// Mitsubishi GX Works2 project: blood pressure test   PLC: FX3G

// global labels: Global1
VAR_GLOBAL
  start_machine AT X007 : BOOL;
  take_test AT X000 : BOOL;
  took_pill AT X001 : BOOL;
  timer_for_gap AT TS1 : BOOL;
  first_test AT D8280 : INT;
  second_test AT D8281 : INT;
  machine_on AT Y007 : BOOL;
  high_blood_pressure AT Y002 : BOOL;
  time_for_next_test AT Y004 : BOOL;
END_VAR
VAR_GLOBAL CONSTANT
  time_to_wait : INT := 50;
END_VAR
VAR_GLOBAL
  took_first_test AT M0 : BOOL;
  test_finish AT M1 : BOOL;
  end_plan AT X006 : BOOL;
  timer AT TC1 : BOOL;
END_VAR
VAR_GLOBAL CONSTANT
  high : INT := 3200;  (* ד *)
END_VAR
VAR_GLOBAL
  hold_light AT M2 : BOOL;
END_VAR

// task Task_01 (event TRUE, interval 0, priority 31): POU_01

PROGRAM POU_01
(* structured ladder/FBD written out as ST: instructions are called as NAME(EN, inputs, outputs); _pN, _eN, _tN stand for wires *)
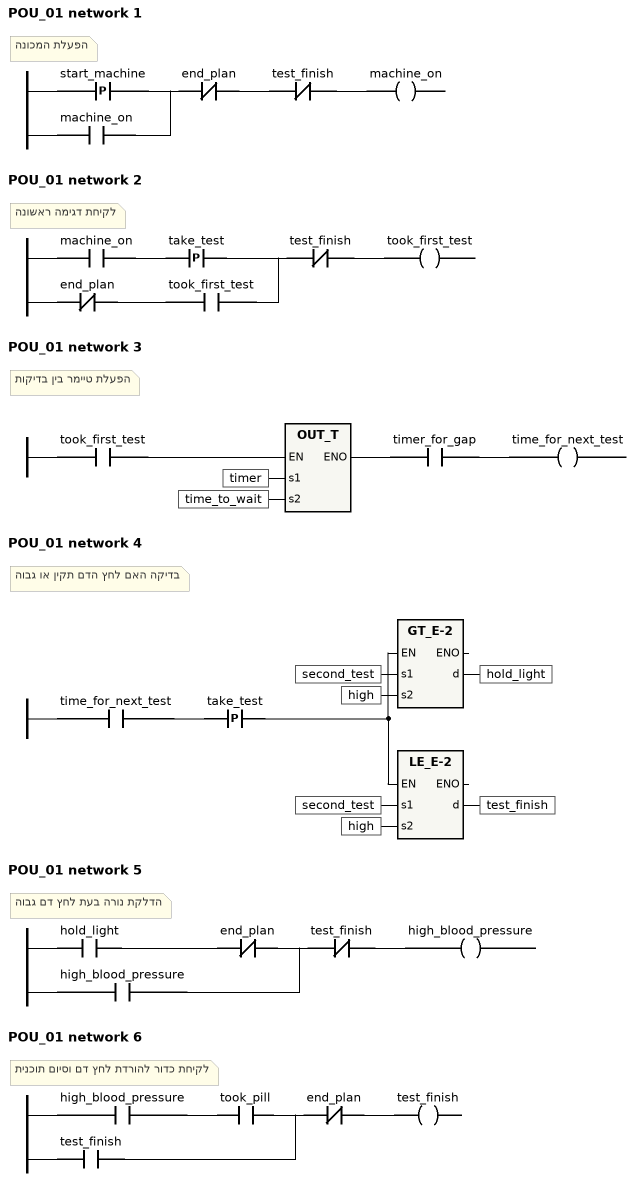
(* network 1 *)
(* הפעלת המכונה *)
machine_on := ((LDP(TRUE, start_machine) OR machine_on) AND NOT end_plan) AND NOT test_finish;
(* network 2 *)
(* לקיחת דגימה ראשונה *)
took_first_test := ((machine_on AND LDP(TRUE, take_test)) OR (NOT end_plan AND took_first_test)) AND NOT test_finish;
(* network 3 *)
(* הפעלת טיימר בין בדיקות *)
_e1 := OUT_T(took_first_test, timer, time_to_wait);
time_for_next_test := _e1 AND timer_for_gap;
(* network 4 *)
(* בדיקה האם לחץ הדם תקין או גבוה *)
_p1 := time_for_next_test AND LDP(TRUE, take_test);
GT_E(_p1, second_test, high, hold_light);
LE_E(_p1, second_test, high, test_finish);
(* network 5 *)
(* הדלקת נורה בעת לחץ דם גבוה *)
high_blood_pressure := ((hold_light AND NOT end_plan) OR high_blood_pressure) AND NOT test_finish;
(* network 6 *)
(* לקיחת כדור להורדת לחץ דם וסיום תוכנית *)
test_finish := ((high_blood_pressure AND took_pill) OR test_finish) AND NOT end_plan;
END_PROGRAM
